(* PLC project SafeLOGIC-1, BrAutomation SafeDESIGNER  4.3.4.4 *)
(* stored: companyURL http://www.br-automation.com, creationDateTime Thu Jun 24 15:38:54 2021 *)

PROGRAM Main
  VAR  (* added by the conversion: wires and edge detectors of the diagram *)
    _SAFEBOOL_TO_BOOL18_OUT : BOOL;
  END_VAR

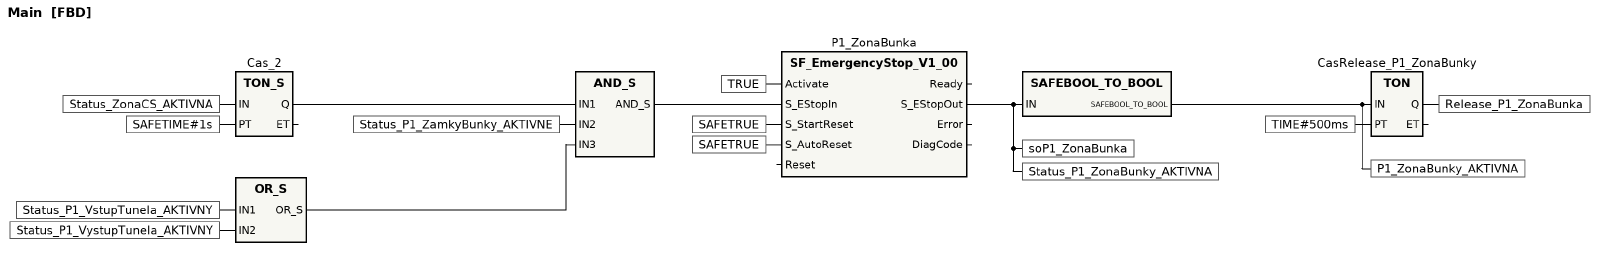
(* FBD diagram, written out as Structured Text *)
Cas_2(IN := Status_ZonaCS_AKTIVNA, PT := SAFETIME#1s);
P1_ZonaBunka(Activate := TRUE, S_EStopIn := AND_S(Cas_2.Q, Status_P1_ZamkyBunky_AKTIVNE, OR_S(Status_P1_VstupTunela_AKTIVNY, Status_P1_VystupTunela_AKTIVNY)), S_StartReset := SAFETRUE, S_AutoReset := SAFETRUE);
soP1_ZonaBunka := P1_ZonaBunka.S_EStopOut;
Status_P1_ZonaBunky_AKTIVNA := P1_ZonaBunka.S_EStopOut;
_SAFEBOOL_TO_BOOL18_OUT := SAFEBOOL_TO_BOOL(P1_ZonaBunka.S_EStopOut);
P1_ZonaBunky_AKTIVNA := _SAFEBOOL_TO_BOOL18_OUT;
CasRelease_P1_ZonaBunky(IN := _SAFEBOOL_TO_BOOL18_OUT, PT := TIME#500ms);
Release_P1_ZonaBunka := CasRelease_P1_ZonaBunky.Q;
END_PROGRAM
